// TIA Portal V16 export
// export: Created 2023-08-28T09:37:35.8408503Z, ExportSetting WithDefaults, DisplayName Totally Integrated Automation Portal, DisplayVersion V16 Update 6, DisplayName TIA Portal Version Control Interface, DisplayVersion V16 Update 2, DisplayName TIA Portal Openness, DisplayVersion V16 Update 6, DisplayName STEP 7 Professional, DisplayVersion V16 Update 6, DisplayName STEP 7 Safety, DisplayVersion V16, DisplayName WinCC Advanced, DisplayVersion V16 Update 6
DATA_BLOCK "V_SoftwareError"   // DB109
{ S7_Optimized_Access := 'TRUE' }
VERSION : 0.1
// stored: AutoNumber false, DBAccessibleFromOPCUA true, IsOnlyStoredInLoadMemory false, IsRetainMemResEnabled false, IsWriteProtectedInAS false, MemoryReserve 0
   VAR
      SoftwareFunctions : Bool;   // //Error is appear in called function
      GetErrorFunction : Bool;   // //Function GET_ERROR() return error
      DiagnosticBuffer : Bool;   // //Error is appear in diagnostic buffer
      ResetErrorSoftware : Bool;   // //Variable connected with button in web site
   END_VAR
BEGIN
END_DATA_BLOCK
